TYPE Mat7d : ARRAY[1..7, 1..7] OF LREAL; END_TYPE

(* stored: Version 1.1.0.1, ProductVersion 3.1.4024.12
   DUT Mat7d: Id {d7487be2-fc82-4961-b87e-2055e0658ce4} *)
